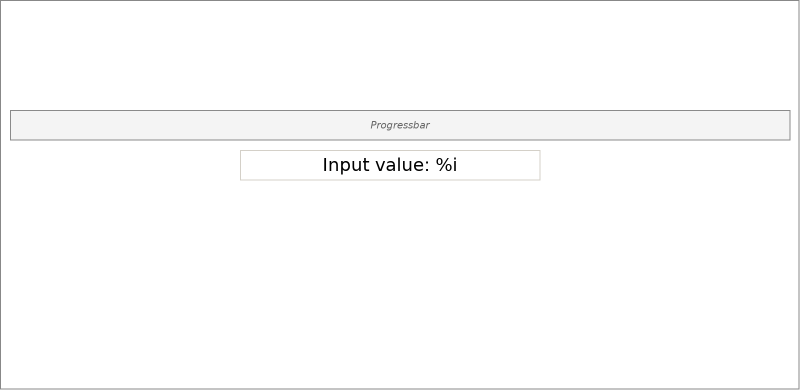
VISUALIZATION VisuAnlogInputControl  // 800x390
VAR_IN_OUT
	pDev : POINTER TO FB_DevAnalogInput;
END_VAR
    Progressbar (10,110 780x30), variable: pDev^.fValue
    Textfield (240,150 300x30), "Input value: %i", text variable: pDev^.fValue
END_VISUALIZATION

(* stored: Version 1.1.0.1, ProductVersion 3.1.4024.11
   Visu VisuAnlogInputControl: Id {2478a7e9-4a11-0395-368d-fa2449d1347a} *)
